FUNCTION_BLOCK FB_Component_ABB_VFD_EIP EXTENDS FB_ComponentBase_SR IMPLEMENTS I_VFD
VAR

    // Outputs
    _ControlWord  AT %Q* : UDINT;
    _EnableMotor  AT %Q* : BOOL;
    _FaultReset   AT %Q* : BOOL;
    _Frequency    AT %Q* : WORD;
    _JogFwd       AT %Q* : BOOL;
    _JogRvs       AT %Q* : BOOL;
    _ReferenceVel AT %Q* : INT;

    // Inputs
    _StatusWord   AT %I* : UDINT;
    _Enabled      AT %I* : BOOL;
    _CommandedVel AT %I* : INT;
    _Faulted      AT %I* : BOOL;
    _Warning      AT %I* : BOOL;
    _FwdActive    AT %I* : BOOL;
    _RvsActive    AT %I* : BOOL;
    _AtSpeed      AT %I* : BOOL;
    _State        AT %I* : USINT;
    // Alarms

    IndicatorAlarms : ARRAY[1..Indicator_ALARMS_COUNT] OF FB_TcAlarm;

    // Internal variables

    Pulse : FB_PulseGenerator;

END_VAR

VAR CONSTANT
    Indicator_ALARMS_COUNT : UDINT := 5;
END_VAR

PROPERTY AtSpeed : bool
GET
AtSpeed := _AtSpeed;
END_GET
END_PROPERTY

PROPERTY CommandedVel : WORD
GET
CommandedVel := INT_TO_WORD(_CommandedVel);
END_GET
END_PROPERTY

//! @summary This method serves as the entry point for all underlying FB logic
METHOD PUBLIC CyclicLogic

//! @description This method should be called cyclically by descendant function blocks by invoking <c>SUPER^.CyclicLogic()</c>.  Alternatively, the contents of this method could be reimplemented entirely in which case a call to this method would not be necessary.
// Initialise Component

IF NOT _InitComplete THEN
    _InitComplete := Initialize();
    RETURN;
END_IF

// Call Super

SUPER^.CyclicLogic();

// Set Current Alarm Severity

_CurrentAlarmSeverity := F_GetMaxSeverityRaised(Alarms := IndicatorAlarms, CurrentSeverity := _CurrentAlarmSeverity);
END_METHOD

METHOD Disable : BOOL
VAR_INPUT
END_VAR
Disable := FALSE;
JogFwd  := FALSE;
JogRvs  := FALSE;

IF FwdActive = FALSE AND RvsActive = FALSE THEN
    Disable := TRUE;
END_IF
END_METHOD

METHOD Enable : BOOL
VAR_INPUT
END_VAR
Enable := FALSE;

IF Enabled = TRUE THEN
    Enable := TRUE;
END_IF
END_METHOD

PROPERTY Enabled : bool
GET
Enabled := _Enabled;
END_GET
END_PROPERTY

PROPERTY Faulted : bool
GET
Faulted := _Faulted;
END_GET
END_PROPERTY

PROPERTY FaultReset : bool
SET
_FaultReset := FaultReset;
END_SET
END_PROPERTY

PROPERTY Frequency : WORD
SET
_Frequency := Frequency;
END_SET
END_PROPERTY

PROPERTY FwdActive : bool
GET
FwdActive := _FwdActive;
END_GET
END_PROPERTY

//! @summary Basic component initialization logic
METHOD PROTECTED Initialize : BOOL;

//! @description This method is called by <c>CyclicLogic()</c> as required
CreateEvents();

IF SUPER^.Initialize() THEN
    Initialize := TRUE;
END_IF
END_METHOD

METHOD Jog : BOOL
VAR_INPUT
    JogFW : BOOL := FALSE;
    JogBW : BOOL := FALSE;
END_VAR
IF JogFW THEN
    Jog    := FALSE;
    JogFwd := TRUE;
    JogRvs := FALSE;

    IF FwdActive AND AtSpeed THEN
        Jog := TRUE;
    END_IF
ELSIF JogBW THEN

    Jog    := FALSE;
    JogFwd := FALSE;
    JogRvs := TRUE;

    IF RvsActive AND AtSpeed THEN
        Jog := TRUE;
    END_IF

END_IF
END_METHOD

PROPERTY JogFwd : bool
SET
_JogFwd := JogFwd;
END_SET
END_PROPERTY

PROPERTY JogRvs : bool
SET
_JogRvs := JogRvs;
END_SET
END_PROPERTY

METHOD PROTECTED Monitoring
VAR_INPUT
END_VAR
SUPER^.Monitoring();
END_METHOD

PROPERTY ReferenceVel : WORD
SET
_ReferenceVel := WORD_TO_INT(ReferenceVel);
END_SET
END_PROPERTY

METHOD Reset : BOOL
Reset := FALSE;

IF Faulted THEN
    FaultReset := TRUE;
ELSE
    FaultReset := FALSE;
    Reset      := TRUE;
END_IF
END_METHOD

PROPERTY RvsActive : bool
GET
RvsActive := _RvsActive;
END_GET
END_PROPERTY

PROPERTY State : USINT
GET
State := _State;
END_GET
END_PROPERTY

METHOD Stop : BOOL
VAR_INPUT
END_VAR
Stop   := FALSE;
JogFwd := FALSE;
JogRvs := FALSE;

IF FwdActive = FALSE AND RvsActive = FALSE THEN
    Stop := TRUE;
END_IF
END_METHOD

PROPERTY Warning : bool
GET
Warning := _Warning;
END_GET
END_PROPERTY

END_FUNCTION_BLOCK

(* stored: Version 1.1.0.1
   POU FB_Component_ABB_VFD_EIP: Id {d7c883d8-9a80-4490-8721-5b49535788c7}, SpecialFunc None
   Folder I_ComponentBase: Id {1a5e26c8-b2f3-48e7-a1bd-08bf41235208}
   Folder I_CyclicFB: Id {eb6a33f2-dab4-4b32-b555-554d2e528154}
   Folder I_Template: Id {183fd5de-6fd6-4094-8b6c-f6a1478630c0}
   Folder Methods: Id {763dc642-d6a3-4de0-8949-b38f716aed4a}
   Folder Properties: Id {fdd6fdc2-f9a5-42e0-808c-d95da9152d52}
   Property AtSpeed: Id {c2da8d17-699a-49f6-af39-a4b992efc0ff}
   Get Get: Id {5abf5cb0-02df-4bf6-b8f0-7bc3ec0179c8}
   Property CommandedVel: Id {b0de3e26-6282-46c9-bd2e-a0eb70bdfe2a}
   Get Get: Id {58167d8f-85e5-4ccf-bdb3-54158f8c1858}
   Method CyclicLogic: Id {d2d3a928-681e-4a83-9ca4-5afec98e3054}
   Method Disable: Id {48a91700-8815-4ae6-9d67-419b3f718794}
   Method Enable: Id {88e8d06a-9202-4435-9e48-dc35cdfd49c5}
   Property Enabled: Id {87b27ac0-90ae-4aac-b832-a4d9894f7c2d}
   Get Get: Id {13a12958-884c-4353-ad98-3dd077b92277}
   Property Faulted: Id {f5d8632e-5de6-4096-b6cd-0707a3edd885}
   Get Get: Id {94df74f0-88ad-4e88-8607-c9eaaff8eade}
   Property FaultReset: Id {57c83385-b413-4b3f-98fe-795a3ecdb97d}
   Set Set: Id {1128f766-22d8-4f5a-aeea-5d71e7c934d6}
   Property Frequency: Id {961a4f44-4f22-42b0-8bf5-04cfe60d005c}
   Set Set: Id {4912c8bb-6b61-45dc-a5f4-dba304dabca4}
   Property FwdActive: Id {934d504a-32b1-4df8-9140-61eb45252847}
   Get Get: Id {096f03ae-9b52-4679-a289-e0bea8f0c2b2}
   Method Initialize: Id {7525ad7f-fedd-4093-afbc-52ff4f72c67d}
   Method Jog: Id {01e5017e-389e-4b57-9256-54bd66bd446e}
   Property JogFwd: Id {f1cf40b1-3c8f-4610-809b-55a9df906e26}
   Set Set: Id {a419c633-e6cb-494b-ac22-dd99adf9bbf6}
   Property JogRvs: Id {90273be1-6d74-44bf-805d-8129fc7bffe1}
   Set Set: Id {2c05e736-3ca6-460a-8afd-51181de40399}
   Method Monitoring: Id {82edacc2-d19c-46ab-8bde-647fb714876b}
   Property ReferenceVel: Id {ca9163a7-2282-4e9c-b50b-f7494123140d}
   Set Set: Id {f2a5b565-e49c-4c88-948f-a598b97020aa}
   Method Reset: Id {a6141c65-1bbe-4d24-acaa-584ea1a1b527}
   Property RvsActive: Id {3b085962-a19d-40a1-8e73-192e429a5b37}
   Get Get: Id {0963eca2-f265-4d35-8393-393bb4ad9a82}
   Property State: Id {90420ee1-1438-4858-bdae-062d1682082d}
   Get Get: Id {6c665aaa-0f49-4427-b603-da46856d721e}
   Method Stop: Id {3cc8b87d-7054-4d0c-bd81-a11eac31a237}
   Property Warning: Id {04d0b7f3-e15b-477e-877e-7f1a39342182}
   Get Get: Id {a1a914df-feb7-4638-85d3-2e4aa1bd6d49} *)
